Fanuc KAREL source: LOAD.kl

PROGRAM T
%NOLOCKGROUP
VAR
 v0 : STRING[40]
 v1 : INTEGER
 v2 : INTEGER
BEGIN
 LOAD(v0, v1, v2)
END T
